TYPE DUT_RECIPE_USERPARAMETEROUTPUT :
STRUCT
	Dummy: BOOL := TRUE;
	Name: STRING(80);
	Description: STRING(80);
	Unit: STRING(80);
	MinValue: LREAL;
	MaxValue: LREAL;
	Default: LREAL;
	Step: LREAL;
END_STRUCT
END_TYPE

(* stored: Version 1.1.0.1, ProductVersion 3.1.0.25
   DUT DUT_RECIPE_USERPARAMETEROUTPUT: Id {56ff042f-ca8a-469c-a937-d8faf3d51916} *)
